FUNCTION_BLOCK FB_HeatPump EXTENDS FB_ActuatorContinous
VAR_INPUT
END_VAR
VAR_OUTPUT
	bError : BOOL;
END_VAR
VAR
	{attribute 'OPC.UA.DA' := '1'}
	localState : ST_HeatPumpState;
	
	//default parameters
	localDefaultParameters : ST_HeatPumpDefaultParameters;
	
	//analog converters
	OutputConverter : FB_AnalogOutput(fUpperLimit := 80, fLowerLimit := 0);
	
	//I/O Links
	nSetPoint_OUT			AT %Q* : INT; //Set position linked to terminal
	bSetStatusOn_OUT 		AT %Q* : BOOL; //SetStatus linked to terminal
	bStatusOn_IN			AT %I* : BOOL; //Error state linked to terminal
	bError_IN 				AT %I* : BOOL; //Error state linked to terminal
END_VAR

MAIN();
OutputConverter(fValue := fSetPoint);

METHOD GetState : BOOL
VAR_INPUT
END_VAR
//local state
controlState.bStatusOn := bStatusOn_IN;
localState.bError := bError_IN;
bStatusOn := controlState.bStatusOn;
bError := localState.bError;
END_METHOD

METHOD PROTECTED  SetSetPointLimits : BOOL
VAR_INPUT
END_VAR
aSetPointLimits[1] := localDefaultParameters.aSetPointLimitsTemperature[1];
aSetPointLimits[2] := localDefaultParameters.aSetPointLimitsTemperature[2];
END_METHOD

METHOD SetState : BOOL
VAR_INPUT
END_VAR
setPointState.fSetPoint := fSetPoint;
setPointState.aSetPointLimits := aSetPointLimits;
setPointState.sSetPointUnit := 'degreeC';

nSetPoint_OUT := OutputConverter.nValue;  //converts real setpoint for terminal
bSetStatusOn_OUT := bSetStatusOn;
END_METHOD

PROPERTY ST_DefaultParameters : REFERENCE TO ST_HeatPumpDefaultParameters
GET
ST_DefaultParameters REF= localDefaultParameters;
END_GET
SET
localDefaultParameters := ST_DefaultParameters;
END_SET
END_PROPERTY

END_FUNCTION_BLOCK

(* stored: Version 1.1.0.1, ProductVersion 3.1.4024.10
   POU FB_HeatPump: Id {0dd9755f-94cf-444c-81a9-fd0cdb4903c5}, SpecialFunc None
   Method GetState: Id {60ebd37c-571c-4562-87b5-edba5ef517b1}
   Method SetSetPointLimits: Id {82c7001b-502f-4eed-ad12-bc20db3b7e0a}
   Method SetState: Id {bde501ed-c924-424b-8141-2c77fd6f9860}
   Property ST_DefaultParameters: Id {39d79361-27f7-4837-ba9c-e45ae9ffbf52}
   Get Get: Id {9f6645e9-f40a-4e31-bf3b-642c7cf82de4}
   Set Set: Id {a9cbb37c-f381-4cc5-942a-0cfa78cb8d38} *)
